{attribute 'qualified_only'}
VAR_GLOBAL CONSTANT
	MaxTestCount : DINT := 4;
END_VAR

(* stored: Version 1.1.0.1
   GVL TestSuite_Parameter: Id {71977508-7c74-4ec9-b7a4-3255aee38094}, ParameterList True *)
